// LS Electric XG5000 project: 과년67_1_4
// PLC NewPLC
// module base 0 slot 0: 입출력 모듈:XBC-DR20S (DC 24V 입력 12점, 릴레이 출력 8점)

PROGRAM NewProgram (task: 스캔 프로그램)

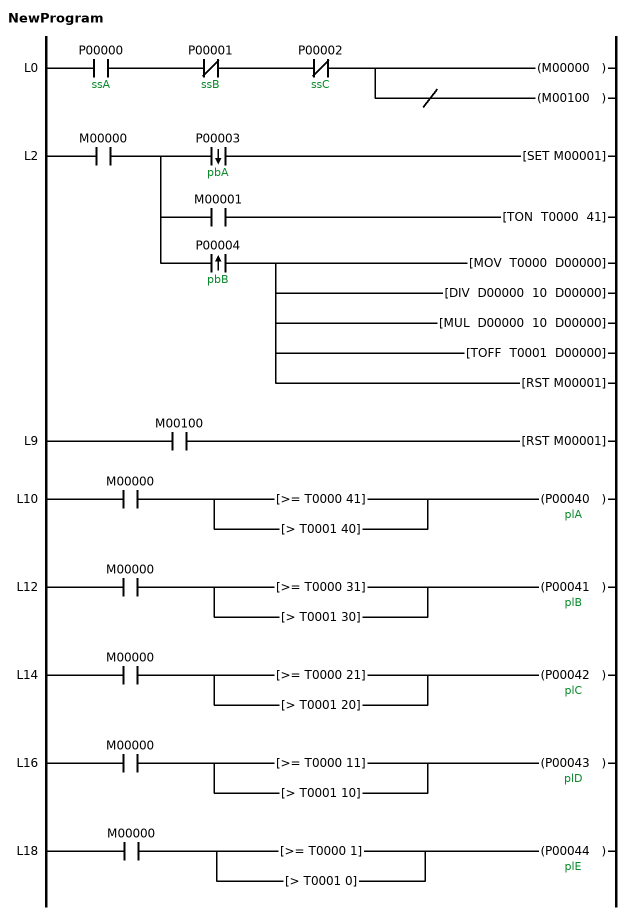
; L0
LOAD      P00000	// ssA
AND NOT   P00001	// ssB
AND NOT   P00002	// ssC
OUT       M00000
NOT
OUT       M00100
; L2
LOAD      M00000
MPUSH
ANDN      P00003	// pbA
SET       M00001
MLOAD
AND       M00001
TON       T0000 41
MPOP
ANDP      P00004	// pbB
MOV       T0000 D00000
DIV       D00000 10 D00000
MUL       D00000 10 D00000
TOFF      T0001 D00000
RST       M00001
; L9
LOAD      M00100
RST       M00001
; L10
LOAD      M00000
LOAD>=    T0000 41
OR>       T0001 40
AND LOAD
OUT       P00040	// plA
; L12
LOAD      M00000
LOAD>=    T0000 31
OR>       T0001 30
AND LOAD
OUT       P00041	// plB
; L14
LOAD      M00000
LOAD>=    T0000 21
OR>       T0001 20
AND LOAD
OUT       P00042	// plC
; L16
LOAD      M00000
LOAD>=    T0000 11
OR>       T0001 10
AND LOAD
OUT       P00043	// plD
; L18
LOAD      M00000
LOAD>=    T0000 1
OR>       T0001 0
AND LOAD
OUT       P00044	// plE

VARIABLES AND COMMENTS (devices not used above)
P00005	BIT	pbC